KUKA KRL program: Reverselooping.src

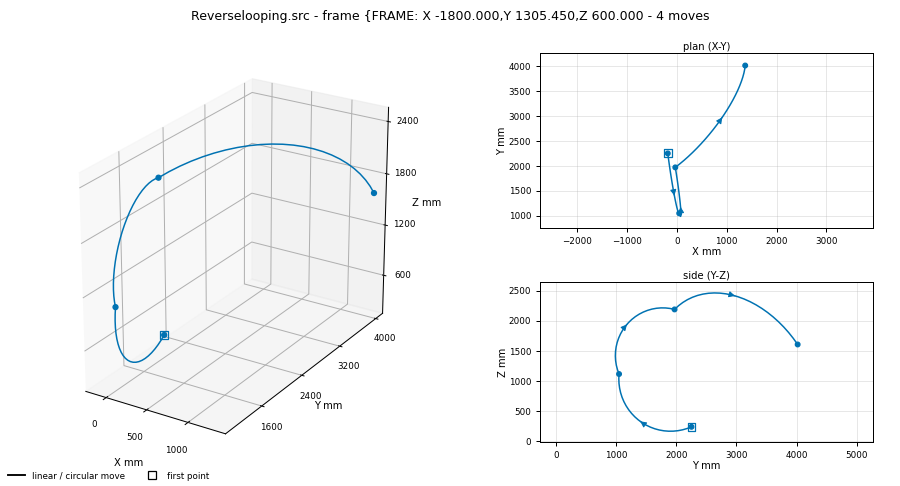
[picture p0: tool path of Reverselooping.src in frame {FRAME: X -1800.000,Y 1305.450,Z 600.000, 4 of 5 moves have a stored position in this frame; points joined in program order, loops and branches not executed]
&ACCESS RVP
&REL 1
&PARAM TEMPLATE = C:\KRC\Roboter\Template\vorgabe
&PARAM EDITMASK = *
DEF Reverselooping ( )
EXT BAS (BAS_COMMAND :IN,REAL :IN )


; GLOBAL INTERRUPT DECL 3 WHEN $STOPMESS==TRUE DO IR_STOPM ( )
; INTERRUPT ON 3

;FOLD Initialise and set default speed
BAS (#INITMOV,0)
BAS (#VEL_PTP,100)
BAS (#ACC_PTP,20)
$VEL.CP=0.2
BAS (#TOOL,0)
BAS (#BASE,0)
;ENDFOLD

;;FOLD STARTPOS
;$BWDSTART = FALSE
;PDAT_ACT = PDEFAULT
;BAS(#PTP_DAT)
;FDAT_ACT = {TOOL_NO 0,BASE_NO 0,IPO_FRAME #BASE}
;BAS(#FRAMES)
;;ENDFOLD

$ADVANCE = 5

;FOLD ---- Quickly skip BCO ----
; PTP $AXIS_ACT
;ENDFOLD

;FOLD ---- GO HOME ----
; PTP {A1 0.000, A2 -90.000, A3 90.000, A4 0.000, A5 0.000, A6 0.000, E1 0, E2 0, E3 0, E4 0, E5 0, E6 0}
;ENDFOLD


; Program generated by RoboDK v5.9.5 for KUKA KR 150 L120/2 on 12/01/2026 20:43:53
; Using nominal kinematics.
; ---- Setting reference (Base) ----
; BASE_DATA[2] = {FRAME: X -1800.000,Y 1305.450,Z 600.000,A -90.000,B 0.000,C 0.000}
$BASE = {FRAME: X -1800.000,Y 1305.450,Z 600.000,A -90.000,B 0.000,C 0.000}
; $BASE = BASE_DATA[2]
; --------------------------
; ---- Setting tool (TCP) ----
$TOOL = {FRAME: X 0.000,Y 0.000,Z 200.000,A 0.000,B 0.000,C 0.000}
; --------------------------
LIN {X -183.063,Y 2254.590,Z 241.349,A -81.380,B -1.565,C 176.848}
CIRC {X -4.078,Y 1182.800,Z 567.456,A -76.437,B -57.871,C 174.068},{X 46.246,Y 1051.750,Z 1118.220,A 87.312,B -74.205,C 11.651}
CIRC {X 79.900,Y 1070.090,Z 1772.210,A 98.021,B -9.241,C 3.192},{X -32.337,Y 1973.530,Z 2191.340,A 105.330,B 65.052,C 34.881}
CIRC {X 768.939,Y 2783.950,Z 2456.380,A -172.755,B 60.901,C 132.978},{X 1371.290,Y 4018.290,Z 1609.120,A -148.331,B 40.155,C 152.256}
PTP {A1 -27.73790,A2 -54.67830,A3 100.89100,A4 -171.55600,A5 46.52490,A6 174.16800}
END
